{attribute 'GeneratedUsingTerminal: AT2050-0500-0021'}
{attribute addProperty BoxType "AT2050-0500-0021"}
{attribute addProperty Id "A_0092_AT2020_5250_0018_AT2020_5250AT2020_01D6DEDF80"}
{attribute addProperty CRC "3616080997"}
{attribute addProperty Size "80"}
TYPE A_0052_AT2050_0500_0021_D7890465 EXTENDS AT2050_86175B41 :
STRUCT
	{attribute addProperty Name "A_0092_AT2020_5250_0018_AT2020_5250"}
	{attribute addProperty PreviousPort "A_0052(AT2050-0500-0021) : B"}
	A_0092_AT2020_5250_0018_AT2020_5250 : AT2020_01D6DEDF;
END_STRUCT
END_TYPE

(* stored: Version 1.2.0.0, ProductVersion 3.1.4024.9
   DUT A_0052_AT2050_0500_0021_D7890465: Id {b5f1d496-ea62-44cf-8653-4e33a9e4f1cf} *)
